FUNCTION_BLOCK FB_SaMElementStarting EXTENDS FB_SaMElement
VAR
END_VAR

END_FUNCTION_BLOCK

(* stored: Version 1.1.0.1
   POU FB_SaMElementStarting: Id {1c659e13-4213-0840-3d68-6ca3a903e38a}, SpecialFunc None *)
